// TIA Portal V16 export
// export: Created 2023-03-29T11:03:44.5177955Z, ExportSetting WithDefaults, DisplayName Totally Integrated Automation Portal, DisplayVersion V16 Update 6, DisplayName TIA Portal Version Control Interface, DisplayVersion V16 Update 2, DisplayName TIA Portal Openness, DisplayVersion V16 Update 6, DisplayName STEP 7 Professional, DisplayVersion V16 Update 6, DisplayName STEP 7 Safety, DisplayVersion V16, DisplayName WinCC Advanced, DisplayVersion V16 Update 6
VAR_GLOBAL   // PLC tag table "Z1"
   Hbit_Zamknij_Z1 AT %M10.5 : Bool;
   Hbit_Alarm_Z1 AT %M10.0 : Bool;
   CMD_Awaria_Z_1 AT %M52.0 : Bool;   // Awaria zbiorcza
   inputAumaawariaZ_1 AT %M51.2 : Bool;   // znacznik wejście
   Hbit_Otwarta_Z1 AT %M10.1 : Bool;
   Hbit_Zamknieta_Z1 AT %M10.3 : Bool;
   Byte_Status_Z1 AT %MW10 : Word;   // Słowo statusu napędu
   inputAumagotowośćZ_1 AT %M51.1 : Bool;   // znacznik wejście
   inputAwariaMomentZ_1 AT %M50.6 : Bool;   // znacznik wejście
   isGotowość_Z_1 AT %M50.0 : Bool;   // bit gotowości wspólny
   Hbit_Auto_Manu_Z1 AT %M10.7 : Bool;
   Hbit_Reset_Z1 AT %M10.6 : Bool;
   inputOtwartaZ_1 AT %M50.2 : Bool;   // znacznik wejście
   inputAumalokalneZ_1 AT %M50.7 : Bool;   // znacznik wejście
   setSVMC_Z_1 AT %M51.4 : Bool;   // Znacznik polecenia zamknij w trybie automat
   Hbit_REN_Z1 AT %M10.2 : Bool;
   setAlarm_Moment_Z_1 AT %M51.5 : Bool;   // znacznik alarmu od momentówki w trybie zdalnym (aut/mamnual)
   inputAumaautomatZ_1 AT %M51.0 : Bool;   // znacznik wejście
   inputRuch_Z_1 AT %M50.5 : Bool;   // znacznik wejście
   CMD_Close_Z_1 AT %M51.7 : Bool;   // załącz zamykanie
   inputREMT_Z_1 AT %M50.1 : Bool;   // znacznik wejście zdalne
   CMD_Open_Z_1 AT %M51.6 : Bool;   // załącz otwieranie
   Hbit_Otwórz_Z1 AT %M10.4 : Bool;
   inputZamkniętaZ_1 AT %M50.3 : Bool;   // znacznik wejście
   isAUMA_Z_1 AT %M52.2 : Bool;   // przęłącznik wymiany na AUMA
   setSVMO_Z_1 AT %M51.3 : Bool;   // Znacznik polecenia otwórz w trybie automat
END_VAR
